INTERFACE I_OutputPortVisitor

METHOD VisitOutputPort
VAR_INPUT
	VisitingOutputPort : I_OutputPort;
END_VAR
END_METHOD

END_INTERFACE

(* stored: Version 1.1.0.1, ProductVersion 3.1.4024.12
   Itf I_OutputPortVisitor: Id {8598d448-75ec-4ea6-bc6f-68222ff84725}
   Method VisitOutputPort: Id {0bf119fc-6e60-46c1-b9f9-5f3a0edd4b44} *)
